(* IEC 61131-3 sources: repolevel_ST_code_completion/verifier, 3 files *)

(* ---- test.st ---- *)
FUNCTION_BLOCK TestFB
VAR_INPUT
    x: BOOL;
END_VAR
VAR_OUTPUT
    y: BOOL;
END_VAR
BEGIN
    y := x2221;
    xg = 1;
END_FUNCTION_BLOCK

(* ---- test_1.st ---- *)
FUNCTION_BLOCK TestFB
VAR_INPUT
    x: BOOL;
END_VAR
VAR_OUTPUT
    y: BOOL;
END_VAR
    y := x;
END_FUNCTION_BLOCK

(* ---- test_fixed.st ---- *)
FUNCTION_BLOCK TestFB
VAR_INPUT
    x: BOOL;
END_VAR
VAR_OUTPUT
    y: BOOL;
END_VAR
VAR
    xg: BOOL; // Declare xg properly based on its expected usage or functionality
END_VAR

    y := x;
    xg := TRUE; // Assuming you want to set xg to TRUE

END_FUNCTION_BLOCK
